{attribute 'reflection'} 
FUNCTION_BLOCK AnalogInputREAL IMPLEMENTS I_AnalogChannel
VAR_INPUT
END_VAR
VAR_OUTPUT
END_VAR
VAR
	sIdentifier:				STRING(25);	// Equipment ID
	Channel			AT%I*: REAL;	// Link to input
END_VAR

// https://github.com/PeterZerlauth/Tc3_Component

PROPERTY PUBLIC P_ID : String(25)
GET
P_ID:= sIdentifier;
END_GET
END_PROPERTY

PROPERTY P_State : EPlcMappingStatus
GET
P_State:= F_GetMappingStatus(ADR(Channel), SIZEOF(INT));
END_GET
END_PROPERTY

PROPERTY PUBLIC P_Value : Lreal
GET
P_Value:= Channel;
END_GET
SET // PUBLIC
Channel:= LREAL_TO_INT(P_Value);
END_SET
END_PROPERTY

END_FUNCTION_BLOCK

(* stored: Version 1.1.0.1
   POU AnalogInputREAL: Id {c5681a80-4710-0cb1-013c-9a2c4ca0e165}, SpecialFunc None
   Property P_ID: Id {a1e5cff1-4f73-0d2e-3e16-ce3f636e41a8}
   Get Get: Id {e42a3203-1b5f-064b-1f28-b27bccc29dad}
   Property P_State: Id {e2018757-633b-058a-09a0-400c8f770506}
   Get Get: Id {d0bfb429-c172-0dcb-3376-38b5176b0ccf}
   Property P_Value: Id {711982f6-1bc6-027f-0555-b3e528249a82}
   Get Get: Id {749639a9-b40a-04f7-372b-90c0cf46c5dc}
   Set Set: Id {a71cc7a5-13cb-09b6-21a8-44c832246944} *)
